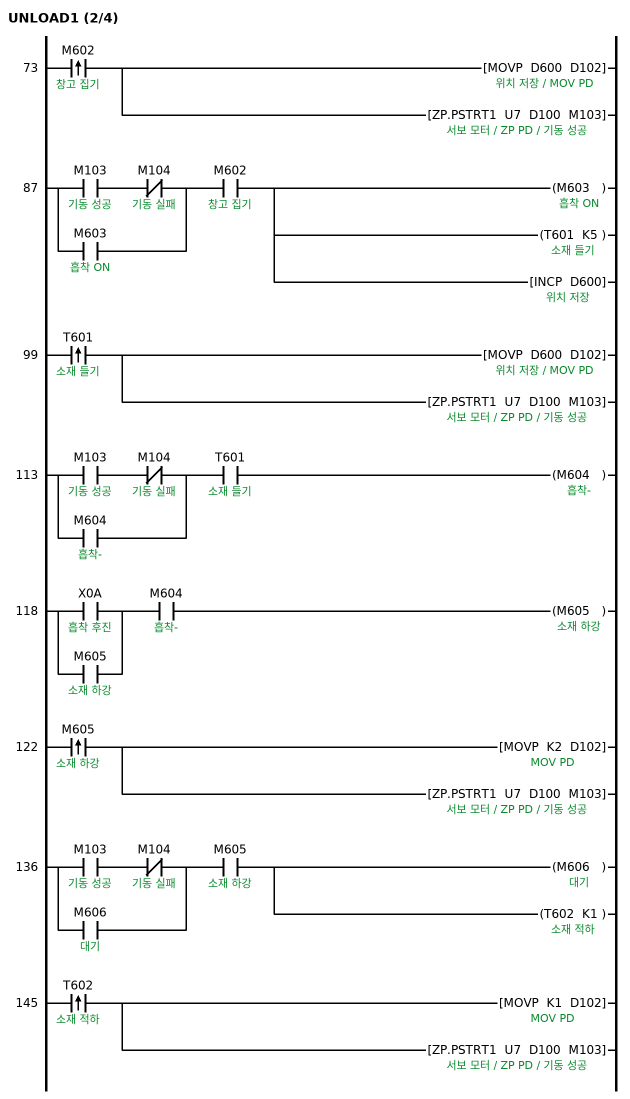
[picture p24: ladder of UNLOAD1, rungs at steps 73 to 145]
73    LDP     M602  ; 창고 집기
      MOVP    D600 D102
      ZP.PSTRT1 U7 D100 M103
87    LD      M103  ; 기동 성공
      ANI     M104  ; 기동 실패
      OR      M603  ; 흡착 ON
      AND     M602  ; 창고 집기
      OUT     M603  ; 흡착 ON
      OUT     T601 K5  ; 소재 들기
      INCP    D600
99    LDP     T601  ; 소재 들기
      MOVP    D600 D102
      ZP.PSTRT1 U7 D100 M103
113   LD      M103  ; 기동 성공
      ANI     M104  ; 기동 실패
      OR      M604  ; 흡착-
      AND     T601  ; 소재 들기
      OUT     M604  ; 흡착-
118   LD      X0A  ; 흡착 후진
      OR      M605  ; 소재 하강
      AND     M604  ; 흡착-
      OUT     M605  ; 소재 하강
122   LDP     M605  ; 소재 하강
      MOVP    K2 D102
      ZP.PSTRT1 U7 D100 M103
136   LD      M103  ; 기동 성공
      ANI     M104  ; 기동 실패
      OR      M606  ; 대기
      AND     M605  ; 소재 하강
      OUT     M606  ; 대기
      OUT     T602 K1  ; 소재 적하
145   LDP     T602  ; 소재 적하
      MOVP    K1 D102
      ZP.PSTRT1 U7 D100 M103
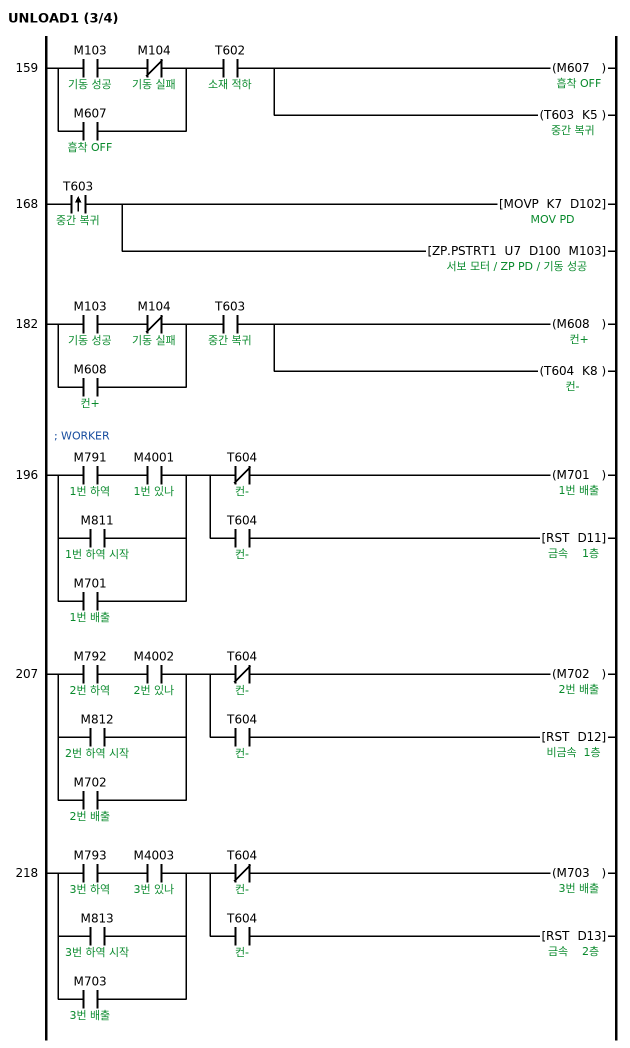
159   LD      M103  ; 기동 성공
      ANI     M104  ; 기동 실패
      OR      M607  ; 흡착 OFF
      AND     T602  ; 소재 적하
      OUT     M607  ; 흡착 OFF
      OUT     T603 K5  ; 중간 복귀
168   LDP     T603  ; 중간 복귀
      MOVP    K7 D102
      ZP.PSTRT1 U7 D100 M103
182   LD      M103  ; 기동 성공
      ANI     M104  ; 기동 실패
      OR      M608  ; 컨+
      AND     T603  ; 중간 복귀
      OUT     M608  ; 컨+
      OUT     T604 K8  ; 컨-
; WORKER
196   LD      M791  ; 1번 하역
      AND     M4001  ; 1번 있나
      OR      M811  ; 1번 하역 시작
      OR      M701  ; 1번 배출
      MPS
      ANI     T604  ; 컨-
      OUT     M701  ; 1번 배출
      MPP
      AND     T604  ; 컨-
      RST     D11  ; 금속    1층
207   LD      M792  ; 2번 하역
      AND     M4002  ; 2번 있나
      OR      M812  ; 2번 하역 시작
      OR      M702  ; 2번 배출
      MPS
      ANI     T604  ; 컨-
      OUT     M702  ; 2번 배출
      MPP
      AND     T604  ; 컨-
      RST     D12  ; 비금속  1층
218   LD      M793  ; 3번 하역
      AND     M4003  ; 3번 있나
      OR      M813  ; 3번 하역 시작
      OR      M703  ; 3번 배출
      MPS
      ANI     T604  ; 컨-
      OUT     M703  ; 3번 배출
      MPP
      AND     T604  ; 컨-
      RST     D13  ; 금속    2층
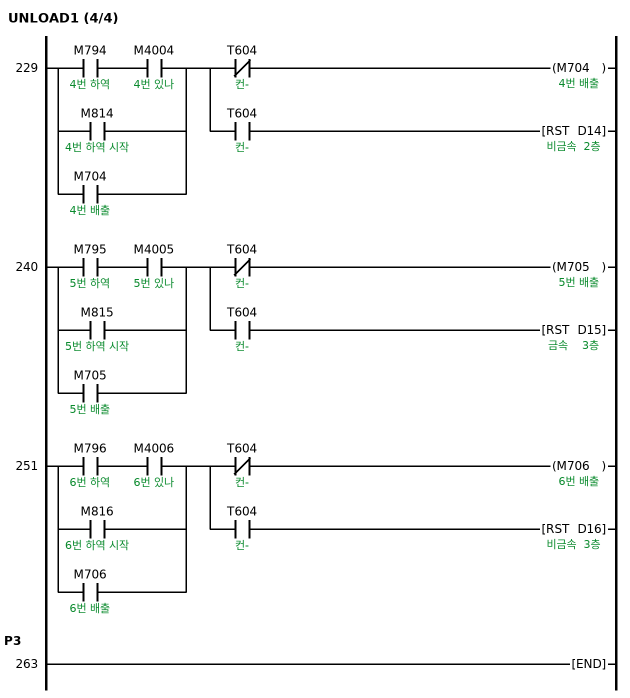
229   LD      M794  ; 4번 하역
      AND     M4004  ; 4번 있나
      OR      M814  ; 4번 하역 시작
      OR      M704  ; 4번 배출
      MPS
      ANI     T604  ; 컨-
      OUT     M704  ; 4번 배출
      MPP
      AND     T604  ; 컨-
      RST     D14  ; 비금속  2층
240   LD      M795  ; 5번 하역
      AND     M4005  ; 5번 있나
      OR      M815  ; 5번 하역 시작
      OR      M705  ; 5번 배출
      MPS
      ANI     T604  ; 컨-
      OUT     M705  ; 5번 배출
      MPP
      AND     T604  ; 컨-
      RST     D15  ; 금속    3층
251   LD      M796  ; 6번 하역
      AND     M4006  ; 6번 있나
      OR      M816  ; 6번 하역 시작
      OR      M706  ; 6번 배출
      MPS
      ANI     T604  ; 컨-
      OUT     M706  ; 6번 배출
      MPP
      AND     T604  ; 컨-
      RST     D16  ; 비금속  3층
      P3
263   END
END_PROGRAM

PROGRAM CONFIG
0     END
END_PROGRAM

// device comments not shown above
X0C  ; 흡착 여부
X17  ; PB3
X18  ; PB4
X1B  ; PB7
X1C  ; Toggle
M8  ; 금속임
M9  ; 판별됨
T0  ; 소재 없음
T5  ; 내리기
T6  ; 올리기
D1502  ; 에러 리셋
